Xinje XDPPro project, PLC1: XD5-60T10 (software 3.7.14b 2022-06-24)

PROGRAM 梯形图

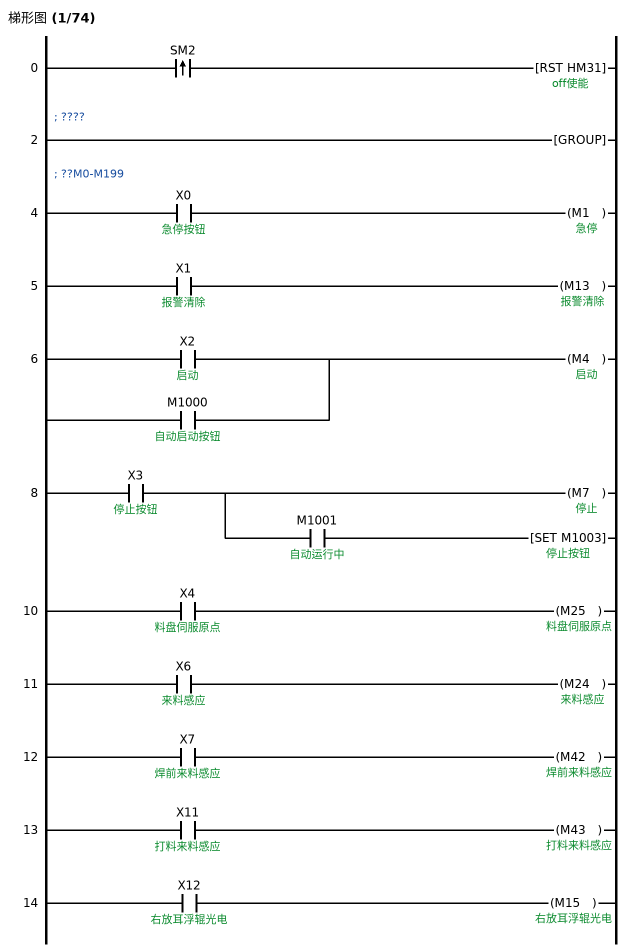
LDP    SM2
RST    HM31	; off使能
; ????
GROUP
; ??M0-M199
LD     X0	; 急停按钮
OUT    M1	; 急停
LD     X1	; 报警清除
OUT    M13	; 报警清除
LD     X2	; 启动
OR     M1000	; 自动启动按钮
OUT    M4	; 启动
LD     X3	; 停止按钮
OUT    M7	; 停止
AND    M1001	; 自动运行中
SET    M1003	; 停止按钮
LD     X4	; 料盘伺服原点
OUT    M25	; 料盘伺服原点
LD     X6	; 来料感应
OUT    M24	; 来料感应
LD     X7	; 焊前来料感应
OUT    M42	; 焊前来料感应
LD     X11	; 打料来料感应
OUT    M43	; 打料来料感应
LD     X12	; 右放耳浮辊光电
OUT    M15	; 右放耳浮辊光电

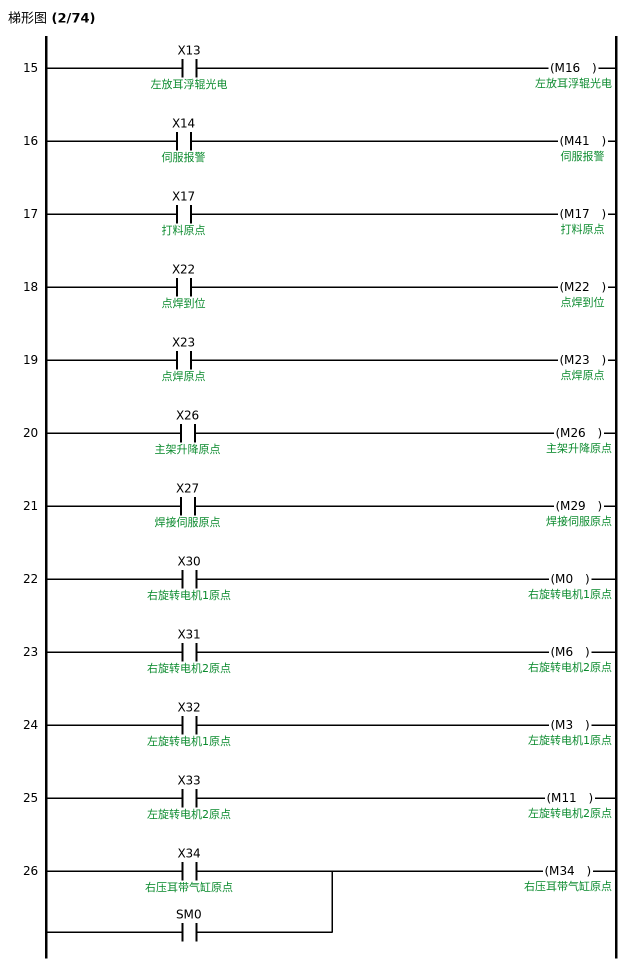
LD     X13	; 左放耳浮辊光电
OUT    M16	; 左放耳浮辊光电
LD     X14	; 伺服报警
OUT    M41	; 伺服报警
LD     X17	; 打料原点
OUT    M17	; 打料原点
LD     X22	; 点焊到位
OUT    M22	; 点焊到位
LD     X23	; 点焊原点
OUT    M23	; 点焊原点
LD     X26	; 主架升降原点
OUT    M26	; 主架升降原点
LD     X27	; 焊接伺服原点
OUT    M29	; 焊接伺服原点
LD     X30	; 右旋转电机1原点
OUT    M0	; 右旋转电机1原点
LD     X31	; 右旋转电机2原点
OUT    M6	; 右旋转电机2原点
LD     X32	; 左旋转电机1原点
OUT    M3	; 左旋转电机1原点
LD     X33	; 左旋转电机2原点
OUT    M11	; 左旋转电机2原点
LD     X34	; 右压耳带气缸原点
OR     SM0
OUT    M34	; 右压耳带气缸原点

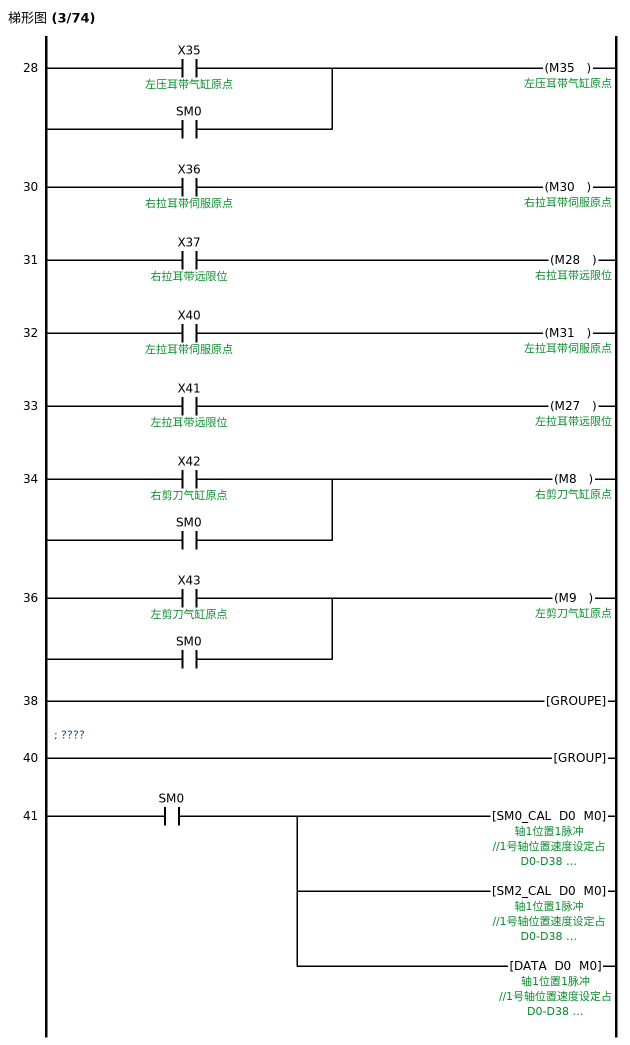
LD     X35	; 左压耳带气缸原点
OR     SM0
OUT    M35	; 左压耳带气缸原点
LD     X36	; 右拉耳带伺服原点
OUT    M30	; 右拉耳带伺服原点
LD     X37	; 右拉耳带远限位
OUT    M28	; 右拉耳带远限位
LD     X40	; 左拉耳带伺服原点
OUT    M31	; 左拉耳带伺服原点
LD     X41	; 左拉耳带远限位
OUT    M27	; 左拉耳带远限位
LD     X42	; 右剪刀气缸原点
OR     SM0
OUT    M8	; 右剪刀气缸原点
LD     X43	; 左剪刀气缸原点
OR     SM0
OUT    M9	; 左剪刀气缸原点
GROUPE
; ????
GROUP
LD     SM0
SM0_CAL D0 M0	; 轴1位置1脉冲   //1号轴位置速度设定占D0-D38 / 右旋转电机1原点
SM2_CAL D0 M0	; 轴1位置1脉冲   //1号轴位置速度设定占D0-D38 / 右旋转电机1原点
DATA   D0 M0	; 轴1位置1脉冲   //1号轴位置速度设定占D0-D38 / 右旋转电机1原点

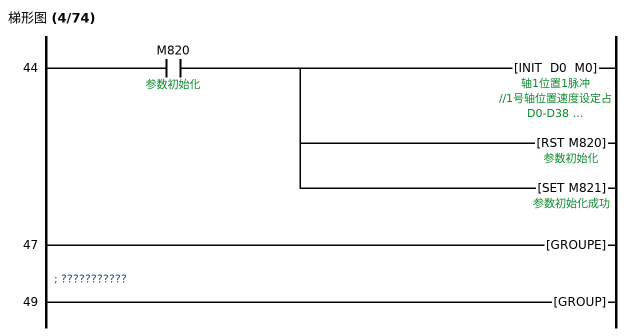
LD     M820	; 参数初始化
INIT   D0 M0	; 轴1位置1脉冲   //1号轴位置速度设定占D0-D38 / 右旋转电机1原点
RST    M820	; 参数初始化
SET    M821	; 参数初始化成功
GROUPE
; ???????????
GROUP

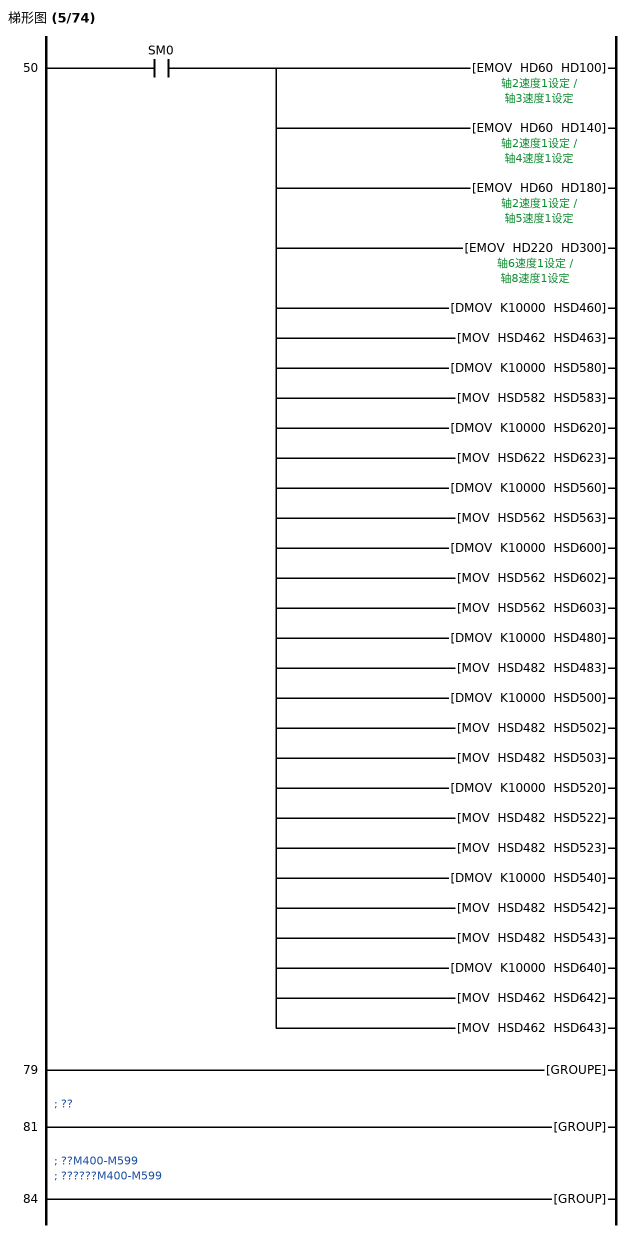
LD     SM0
EMOV   HD60 HD100	; 轴2速度1设定 / 轴3速度1设定
EMOV   HD60 HD140	; 轴2速度1设定 / 轴4速度1设定
EMOV   HD60 HD180	; 轴2速度1设定 / 轴5速度1设定
EMOV   HD220 HD300	; 轴6速度1设定 / 轴8速度1设定
DMOV   K10000 HSD460
MOV    HSD462 HSD463
DMOV   K10000 HSD580
MOV    HSD582 HSD583
DMOV   K10000 HSD620
MOV    HSD622 HSD623
DMOV   K10000 HSD560
MOV    HSD562 HSD563
DMOV   K10000 HSD600
MOV    HSD562 HSD602
MOV    HSD562 HSD603
DMOV   K10000 HSD480
MOV    HSD482 HSD483
DMOV   K10000 HSD500
MOV    HSD482 HSD502
MOV    HSD482 HSD503
DMOV   K10000 HSD520
MOV    HSD482 HSD522
MOV    HSD482 HSD523
DMOV   K10000 HSD540
MOV    HSD482 HSD542
MOV    HSD482 HSD543
DMOV   K10000 HSD640
MOV    HSD462 HSD642
MOV    HSD462 HSD643
GROUPE
; ??
GROUP
; ??M400-M599
; ??????M400-M599
GROUP

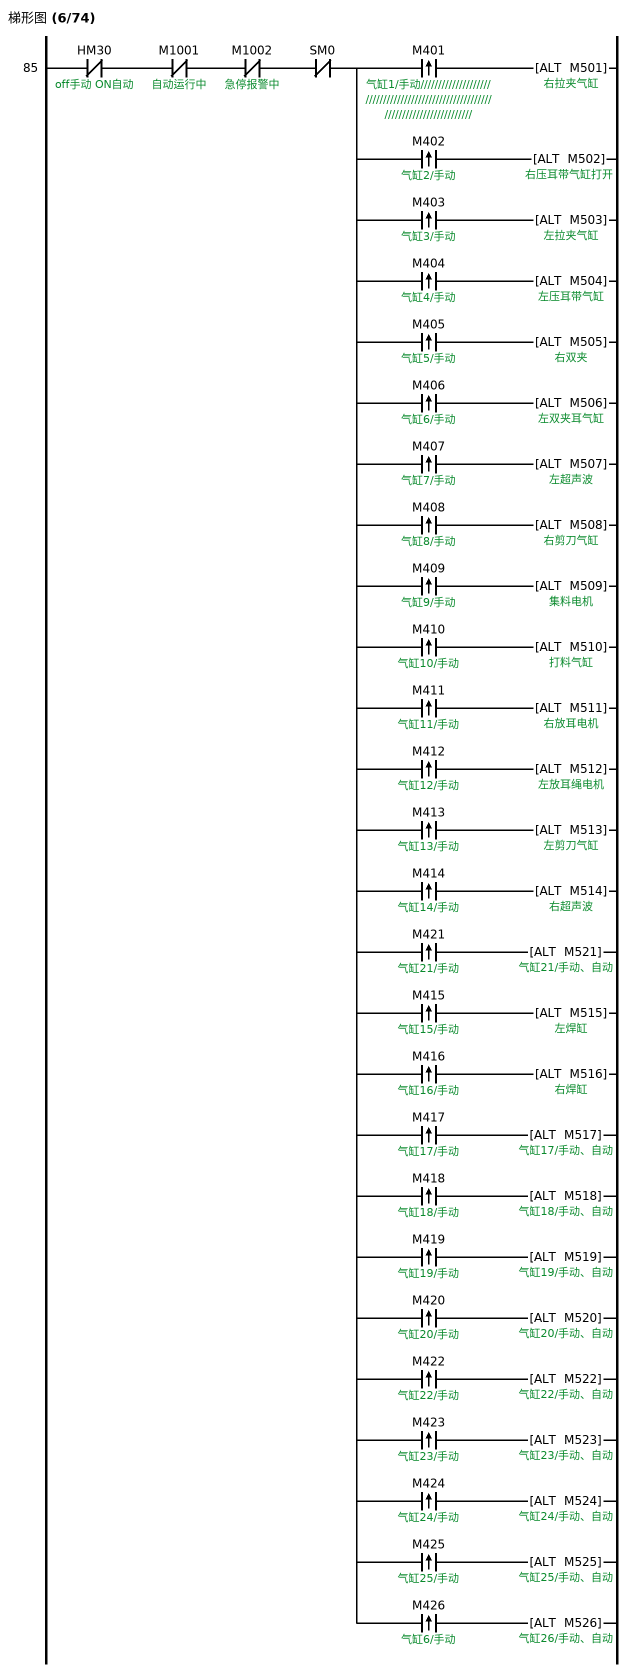
LDI    HM30	; off手动 ON自动
ANI    M1001	; 自动运行中
ANI    M1002	; 急停报警中
ANI    SM0
MPS
ANDP   M401	; 气缸1/手动/////////////////////////////////////////////////////////////////////////////////
ALT    M501	; 右拉夹气缸
MRD
ANDP   M402	; 气缸2/手动
ALT    M502	; 右压耳带气缸打开
MRD
ANDP   M403	; 气缸3/手动
ALT    M503	; 左拉夹气缸
MRD
ANDP   M404	; 气缸4/手动
ALT    M504	; 左压耳带气缸
MRD
ANDP   M405	; 气缸5/手动
ALT    M505	; 右双夹
MRD
ANDP   M406	; 气缸6/手动
ALT    M506	; 左双夹耳气缸
MRD
ANDP   M407	; 气缸7/手动
ALT    M507	; 左超声波
MRD
ANDP   M408	; 气缸8/手动
ALT    M508	; 右剪刀气缸
MRD
ANDP   M409	; 气缸9/手动
ALT    M509	; 集料电机
MRD
ANDP   M410	; 气缸10/手动
ALT    M510	; 打料气缸
MRD
ANDP   M411	; 气缸11/手动
ALT    M511	; 右放耳电机
MRD
ANDP   M412	; 气缸12/手动
ALT    M512	; 左放耳绳电机
MRD
ANDP   M413	; 气缸13/手动
ALT    M513	; 左剪刀气缸
MRD
ANDP   M414	; 气缸14/手动
ALT    M514	; 右超声波
MRD
ANDP   M421	; 气缸21/手动
ALT    M521	; 气缸21/手动、自动
MRD
ANDP   M415	; 气缸15/手动
ALT    M515	; 左焊缸
MRD
ANDP   M416	; 气缸16/手动
ALT    M516	; 右焊缸
MRD
ANDP   M417	; 气缸17/手动
ALT    M517	; 气缸17/手动、自动
MRD
ANDP   M418	; 气缸18/手动
ALT    M518	; 气缸18/手动、自动
MRD
ANDP   M419	; 气缸19/手动
ALT    M519	; 气缸19/手动、自动
MRD
ANDP   M420	; 气缸20/手动
ALT    M520	; 气缸20/手动、自动
MRD
ANDP   M422	; 气缸22/手动
ALT    M522	; 气缸22/手动、自动
MRD
ANDP   M423	; 气缸23/手动
ALT    M523	; 气缸23/手动、自动
MRD
ANDP   M424	; 气缸24/手动
ALT    M524	; 气缸24/手动、自动
MRD
ANDP   M425	; 气缸25/手动
ALT    M525	; 气缸25/手动、自动
MPP
ANDP   M426	; 气缸6/手动
ALT    M526	; 气缸26/手动、自动

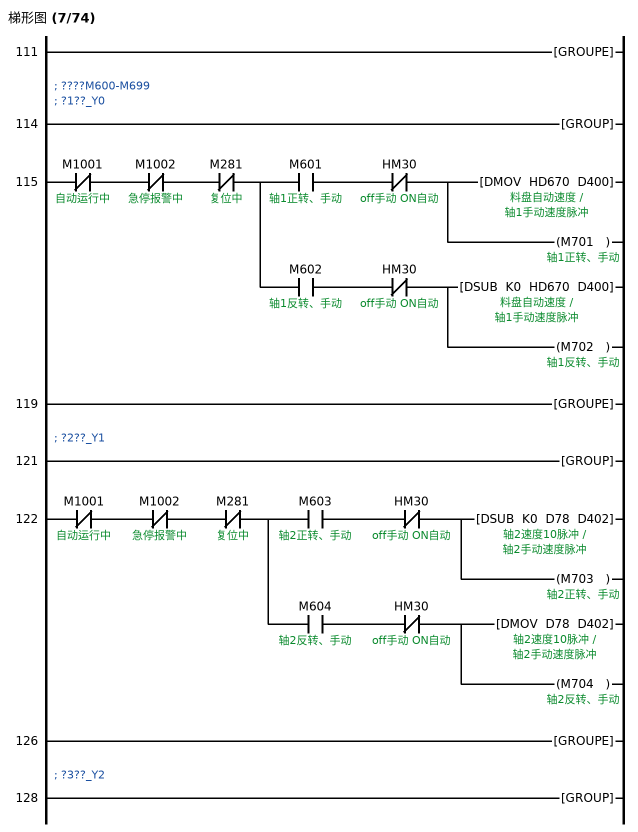
GROUPE
; ????M600-M699
; ?1??_Y0
GROUP
LDI    M1001	; 自动运行中
ANI    M1002	; 急停报警中
ANI    M281	; 复位中
MPS
AND    M601	; 轴1正转、手动
ANI    HM30	; off手动 ON自动
DMOV   HD670 D400	; 料盘自动速度 / 轴1手动速度脉冲
OUT    M701	; 轴1正转、手动
MPP
AND    M602	; 轴1反转、手动
ANI    HM30	; off手动 ON自动
DSUB   K0 HD670 D400	; 料盘自动速度 / 轴1手动速度脉冲
OUT    M702	; 轴1反转、手动
GROUPE
; ?2??_Y1
GROUP
LDI    M1001	; 自动运行中
ANI    M1002	; 急停报警中
ANI    M281	; 复位中
MPS
AND    M603	; 轴2正转、手动
ANI    HM30	; off手动 ON自动
DSUB   K0 D78 D402	; 轴2速度10脉冲 / 轴2手动速度脉冲
OUT    M703	; 轴2正转、手动
MPP
AND    M604	; 轴2反转、手动
ANI    HM30	; off手动 ON自动
DMOV   D78 D402	; 轴2速度10脉冲 / 轴2手动速度脉冲
OUT    M704	; 轴2反转、手动
GROUPE
; ?3??_Y2
GROUP

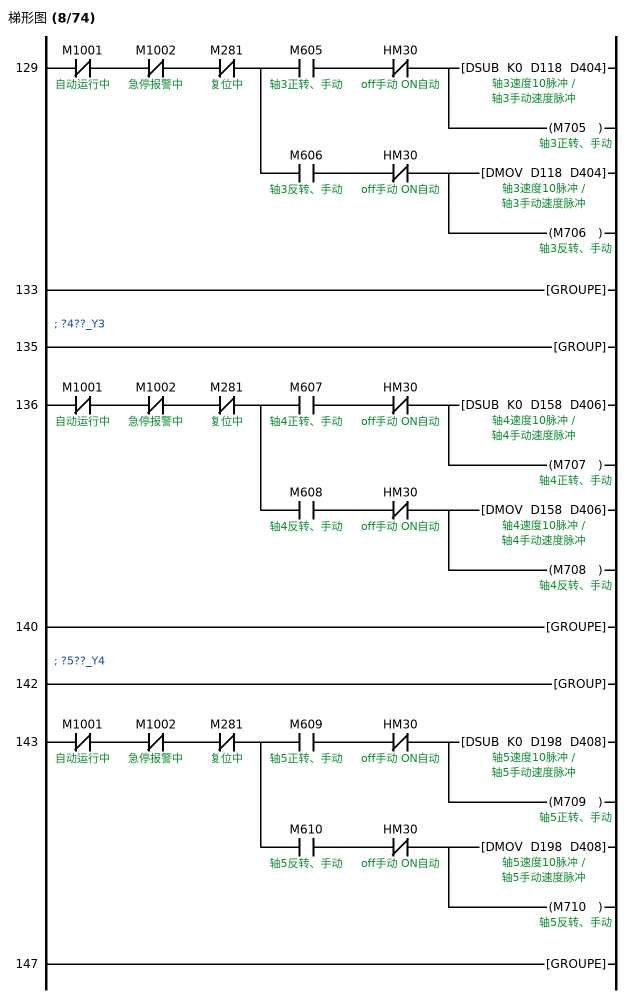
LDI    M1001	; 自动运行中
ANI    M1002	; 急停报警中
ANI    M281	; 复位中
MPS
AND    M605	; 轴3正转、手动
ANI    HM30	; off手动 ON自动
DSUB   K0 D118 D404	; 轴3速度10脉冲 / 轴3手动速度脉冲
OUT    M705	; 轴3正转、手动
MPP
AND    M606	; 轴3反转、手动
ANI    HM30	; off手动 ON自动
DMOV   D118 D404	; 轴3速度10脉冲 / 轴3手动速度脉冲
OUT    M706	; 轴3反转、手动
GROUPE
; ?4??_Y3
GROUP
LDI    M1001	; 自动运行中
ANI    M1002	; 急停报警中
ANI    M281	; 复位中
MPS
AND    M607	; 轴4正转、手动
ANI    HM30	; off手动 ON自动
DSUB   K0 D158 D406	; 轴4速度10脉冲 / 轴4手动速度脉冲
OUT    M707	; 轴4正转、手动
MPP
AND    M608	; 轴4反转、手动
ANI    HM30	; off手动 ON自动
DMOV   D158 D406	; 轴4速度10脉冲 / 轴4手动速度脉冲
OUT    M708	; 轴4反转、手动
GROUPE
; ?5??_Y4
GROUP
LDI    M1001	; 自动运行中
ANI    M1002	; 急停报警中
ANI    M281	; 复位中
MPS
AND    M609	; 轴5正转、手动
ANI    HM30	; off手动 ON自动
DSUB   K0 D198 D408	; 轴5速度10脉冲 / 轴5手动速度脉冲
OUT    M709	; 轴5正转、手动
MPP
AND    M610	; 轴5反转、手动
ANI    HM30	; off手动 ON自动
DMOV   D198 D408	; 轴5速度10脉冲 / 轴5手动速度脉冲
OUT    M710	; 轴5反转、手动
GROUPE

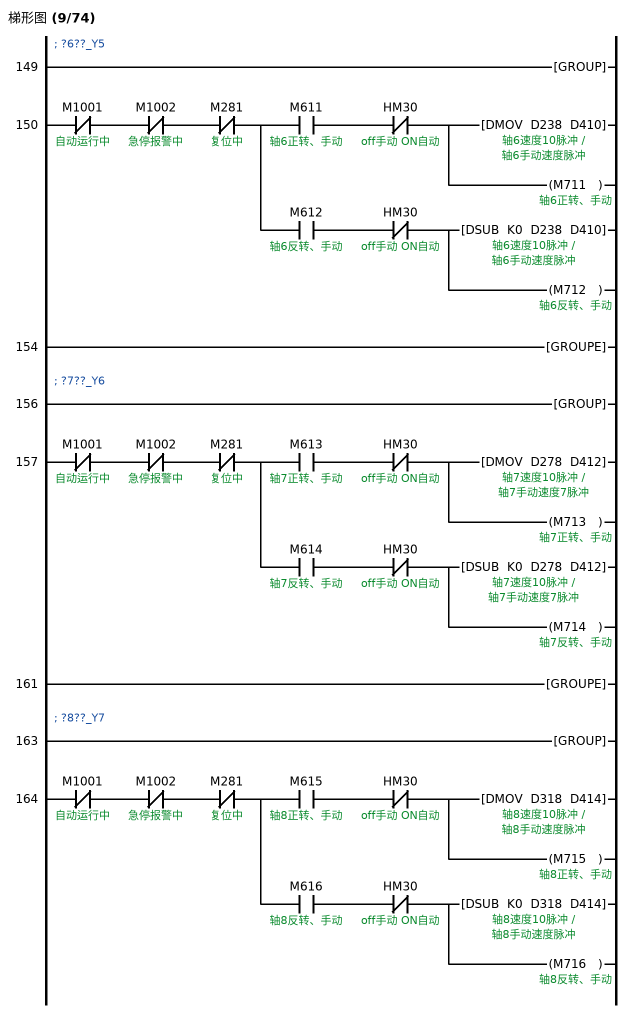
; ?6??_Y5
GROUP
LDI    M1001	; 自动运行中
ANI    M1002	; 急停报警中
ANI    M281	; 复位中
MPS
AND    M611	; 轴6正转、手动
ANI    HM30	; off手动 ON自动
DMOV   D238 D410	; 轴6速度10脉冲 / 轴6手动速度脉冲
OUT    M711	; 轴6正转、手动
MPP
AND    M612	; 轴6反转、手动
ANI    HM30	; off手动 ON自动
DSUB   K0 D238 D410	; 轴6速度10脉冲 / 轴6手动速度脉冲
OUT    M712	; 轴6反转、手动
GROUPE
; ?7??_Y6
GROUP
LDI    M1001	; 自动运行中
ANI    M1002	; 急停报警中
ANI    M281	; 复位中
MPS
AND    M613	; 轴7正转、手动
ANI    HM30	; off手动 ON自动
DMOV   D278 D412	; 轴7速度10脉冲 / 轴7手动速度7脉冲
OUT    M713	; 轴7正转、手动
MPP
AND    M614	; 轴7反转、手动
ANI    HM30	; off手动 ON自动
DSUB   K0 D278 D412	; 轴7速度10脉冲 / 轴7手动速度7脉冲
OUT    M714	; 轴7反转、手动
GROUPE
; ?8??_Y7
GROUP
LDI    M1001	; 自动运行中
ANI    M1002	; 急停报警中
ANI    M281	; 复位中
MPS
AND    M615	; 轴8正转、手动
ANI    HM30	; off手动 ON自动
DMOV   D318 D414	; 轴8速度10脉冲 / 轴8手动速度脉冲
OUT    M715	; 轴8正转、手动
MPP
AND    M616	; 轴8反转、手动
ANI    HM30	; off手动 ON自动
DSUB   K0 D318 D414	; 轴8速度10脉冲 / 轴8手动速度脉冲
OUT    M716	; 轴8反转、手动

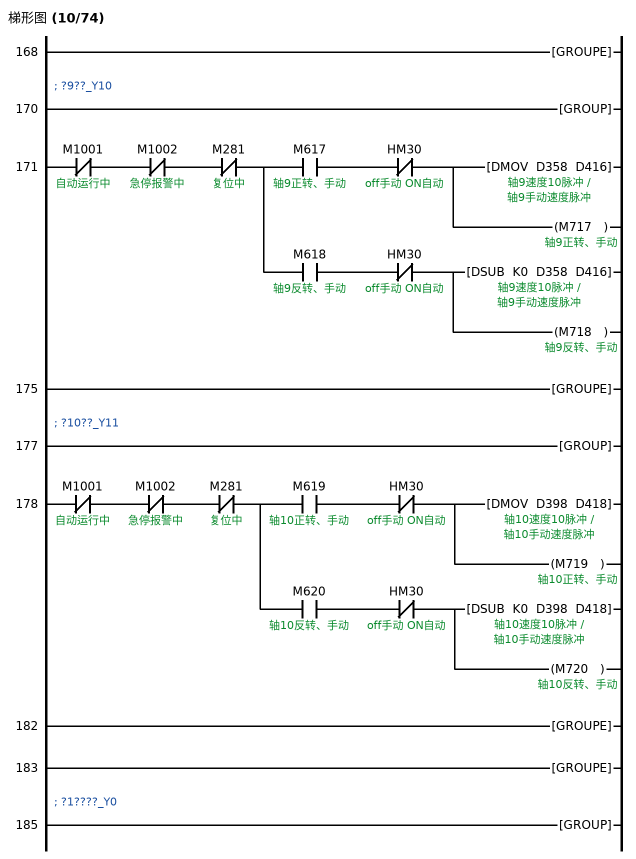
GROUPE
; ?9??_Y10
GROUP
LDI    M1001	; 自动运行中
ANI    M1002	; 急停报警中
ANI    M281	; 复位中
MPS
AND    M617	; 轴9正转、手动
ANI    HM30	; off手动 ON自动
DMOV   D358 D416	; 轴9速度10脉冲 / 轴9手动速度脉冲
OUT    M717	; 轴9正转、手动
MPP
AND    M618	; 轴9反转、手动
ANI    HM30	; off手动 ON自动
DSUB   K0 D358 D416	; 轴9速度10脉冲 / 轴9手动速度脉冲
OUT    M718	; 轴9反转、手动
GROUPE
; ?10??_Y11
GROUP
LDI    M1001	; 自动运行中
ANI    M1002	; 急停报警中
ANI    M281	; 复位中
MPS
AND    M619	; 轴10正转、手动
ANI    HM30	; off手动 ON自动
DMOV   D398 D418	; 轴10速度10脉冲 / 轴10手动速度脉冲
OUT    M719	; 轴10正转、手动
MPP
AND    M620	; 轴10反转、手动
ANI    HM30	; off手动 ON自动
DSUB   K0 D398 D418	; 轴10速度10脉冲 / 轴10手动速度脉冲
OUT    M720	; 轴10反转、手动
GROUPE
GROUPE
; ?1????_Y0
GROUP

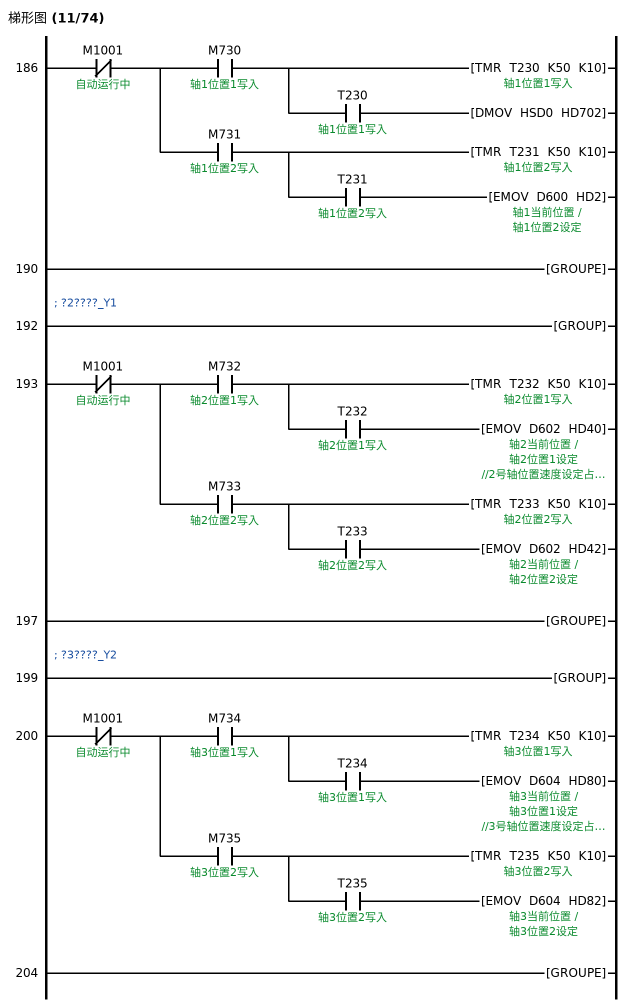
LDI    M1001	; 自动运行中
MPS
AND    M730	; 轴1位置1写入
TMR    T230 K50 K10	; 轴1位置1写入
AND    T230	; 轴1位置1写入
DMOV   HSD0 HD702
MPP
AND    M731	; 轴1位置2写入
TMR    T231 K50 K10	; 轴1位置2写入
AND    T231	; 轴1位置2写入
EMOV   D600 HD2	; 轴1当前位置 / 轴1位置2设定
GROUPE
; ?2????_Y1
GROUP
LDI    M1001	; 自动运行中
MPS
AND    M732	; 轴2位置1写入
TMR    T232 K50 K10	; 轴2位置1写入
AND    T232	; 轴2位置1写入
EMOV   D602 HD40	; 轴2当前位置 / 轴2位置1设定   //2号轴位置速度设定占HD40-HD78
MPP
AND    M733	; 轴2位置2写入
TMR    T233 K50 K10	; 轴2位置2写入
AND    T233	; 轴2位置2写入
EMOV   D602 HD42	; 轴2当前位置 / 轴2位置2设定
GROUPE
; ?3????_Y2
GROUP
LDI    M1001	; 自动运行中
MPS
AND    M734	; 轴3位置1写入
TMR    T234 K50 K10	; 轴3位置1写入
AND    T234	; 轴3位置1写入
EMOV   D604 HD80	; 轴3当前位置 / 轴3位置1设定   //3号轴位置速度设定占HD80-HD118
MPP
AND    M735	; 轴3位置2写入
TMR    T235 K50 K10	; 轴3位置2写入
AND    T235	; 轴3位置2写入
EMOV   D604 HD82	; 轴3当前位置 / 轴3位置2设定
GROUPE

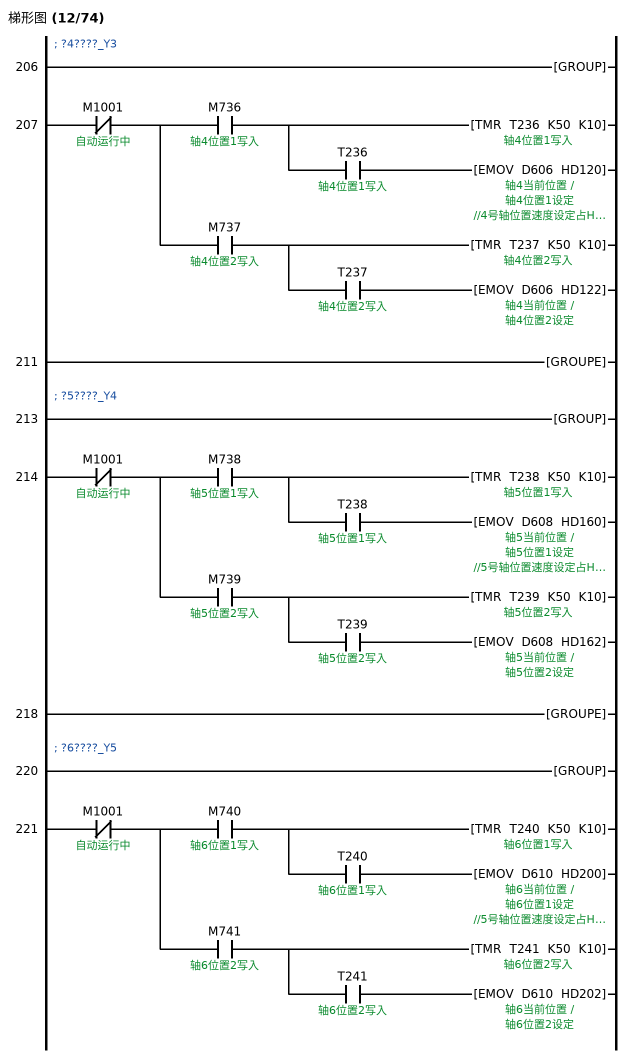
; ?4????_Y3
GROUP
LDI    M1001	; 自动运行中
MPS
AND    M736	; 轴4位置1写入
TMR    T236 K50 K10	; 轴4位置1写入
AND    T236	; 轴4位置1写入
EMOV   D606 HD120	; 轴4当前位置 / 轴4位置1设定   //4号轴位置速度设定占HD120-HD158
MPP
AND    M737	; 轴4位置2写入
TMR    T237 K50 K10	; 轴4位置2写入
AND    T237	; 轴4位置2写入
EMOV   D606 HD122	; 轴4当前位置 / 轴4位置2设定
GROUPE
; ?5????_Y4
GROUP
LDI    M1001	; 自动运行中
MPS
AND    M738	; 轴5位置1写入
TMR    T238 K50 K10	; 轴5位置1写入
AND    T238	; 轴5位置1写入
EMOV   D608 HD160	; 轴5当前位置 / 轴5位置1设定   //5号轴位置速度设定占HD160-HD198
MPP
AND    M739	; 轴5位置2写入
TMR    T239 K50 K10	; 轴5位置2写入
AND    T239	; 轴5位置2写入
EMOV   D608 HD162	; 轴5当前位置 / 轴5位置2设定
GROUPE
; ?6????_Y5
GROUP
LDI    M1001	; 自动运行中
MPS
AND    M740	; 轴6位置1写入
TMR    T240 K50 K10	; 轴6位置1写入
AND    T240	; 轴6位置1写入
EMOV   D610 HD200	; 轴6当前位置 / 轴6位置1设定   //5号轴位置速度设定占HD200-HD238
MPP
AND    M741	; 轴6位置2写入
TMR    T241 K50 K10	; 轴6位置2写入
AND    T241	; 轴6位置2写入
EMOV   D610 HD202	; 轴6当前位置 / 轴6位置2设定

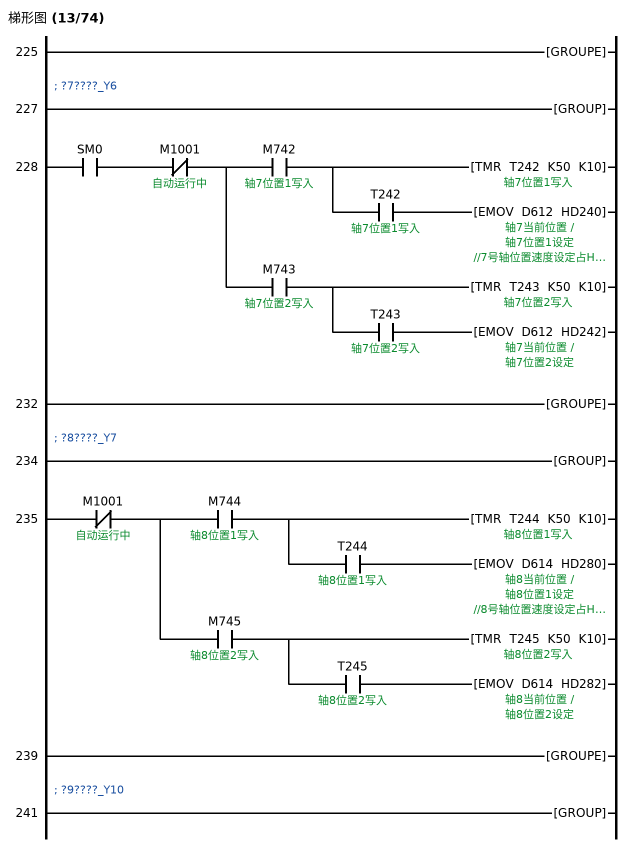
GROUPE
; ?7????_Y6
GROUP
LD     SM0
ANI    M1001	; 自动运行中
MPS
AND    M742	; 轴7位置1写入
TMR    T242 K50 K10	; 轴7位置1写入
AND    T242	; 轴7位置1写入
EMOV   D612 HD240	; 轴7当前位置 / 轴7位置1设定   //7号轴位置速度设定占HD240-HD278
MPP
AND    M743	; 轴7位置2写入
TMR    T243 K50 K10	; 轴7位置2写入
AND    T243	; 轴7位置2写入
EMOV   D612 HD242	; 轴7当前位置 / 轴7位置2设定
GROUPE
; ?8????_Y7
GROUP
LDI    M1001	; 自动运行中
MPS
AND    M744	; 轴8位置1写入
TMR    T244 K50 K10	; 轴8位置1写入
AND    T244	; 轴8位置1写入
EMOV   D614 HD280	; 轴8当前位置 / 轴8位置1设定   //8号轴位置速度设定占HD280-HD318
MPP
AND    M745	; 轴8位置2写入
TMR    T245 K50 K10	; 轴8位置2写入
AND    T245	; 轴8位置2写入
EMOV   D614 HD282	; 轴8当前位置 / 轴8位置2设定
GROUPE
; ?9????_Y10
GROUP

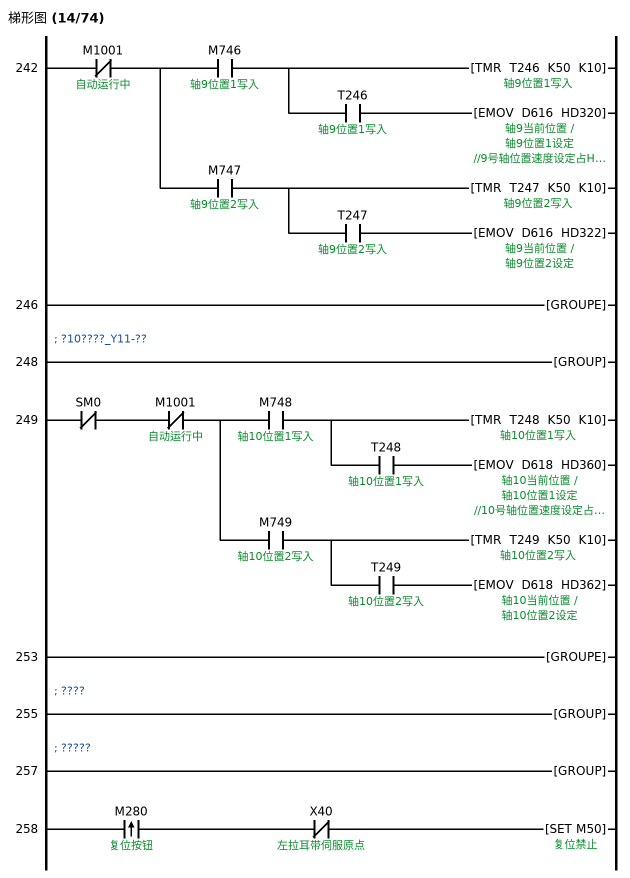
LDI    M1001	; 自动运行中
MPS
AND    M746	; 轴9位置1写入
TMR    T246 K50 K10	; 轴9位置1写入
AND    T246	; 轴9位置1写入
EMOV   D616 HD320	; 轴9当前位置 / 轴9位置1设定   //9号轴位置速度设定占HD320-HD358
MPP
AND    M747	; 轴9位置2写入
TMR    T247 K50 K10	; 轴9位置2写入
AND    T247	; 轴9位置2写入
EMOV   D616 HD322	; 轴9当前位置 / 轴9位置2设定
GROUPE
; ?10????_Y11-??
GROUP
LDI    SM0
ANI    M1001	; 自动运行中
MPS
AND    M748	; 轴10位置1写入
TMR    T248 K50 K10	; 轴10位置1写入
AND    T248	; 轴10位置1写入
EMOV   D618 HD360	; 轴10当前位置 / 轴10位置1设定   //10号轴位置速度设定占HD360-HD398
MPP
AND    M749	; 轴10位置2写入
TMR    T249 K50 K10	; 轴10位置2写入
AND    T249	; 轴10位置2写入
EMOV   D618 HD362	; 轴10当前位置 / 轴10位置2设定
GROUPE
; ????
GROUP
; ?????
GROUP
LDP    M280	; 复位按钮
ANI    X40	; 左拉耳带伺服原点
SET    M50	; 复位禁止

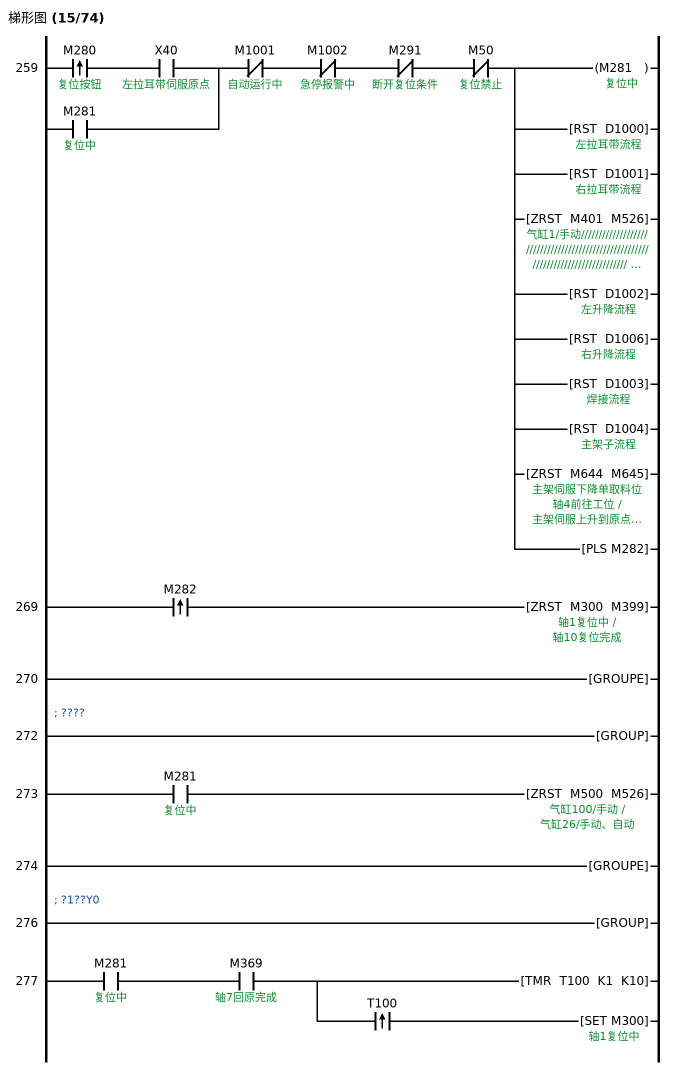
LDP    M280	; 复位按钮
AND    X40	; 左拉耳带伺服原点
OR     M281	; 复位中
ANI    M1001	; 自动运行中
ANI    M1002	; 急停报警中
ANI    M291	; 断开复位条件
ANI    M50	; 复位禁止
OUT    M281	; 复位中
RST    D1000	; 左拉耳带流程
RST    D1001	; 右拉耳带流程
ZRST   M401 M526	; 气缸1/手动///////////////////////////////////////////////////////////////////////////////// / 气缸26/手动、自动
RST    D1002	; 左升降流程
RST    D1006	; 右升降流程
RST    D1003	; 焊接流程
RST    D1004	; 主架子流程
ZRST   M644 M645	; 主架伺服下降单取料位 轴4前往工位 / 主架伺服上升到原点位 轴4前往原点位
PLS    M282
LDP    M282
ZRST   M300 M399	; 轴1复位中 / 轴10复位完成
GROUPE
; ????
GROUP
LD     M281	; 复位中
ZRST   M500 M526	; 气缸100/手动 / 气缸26/手动、自动
GROUPE
; ?1??Y0
GROUP
LD     M281	; 复位中
AND    M369	; 轴7回原完成
TMR    T100 K1 K10
ANDP   T100
SET    M300	; 轴1复位中

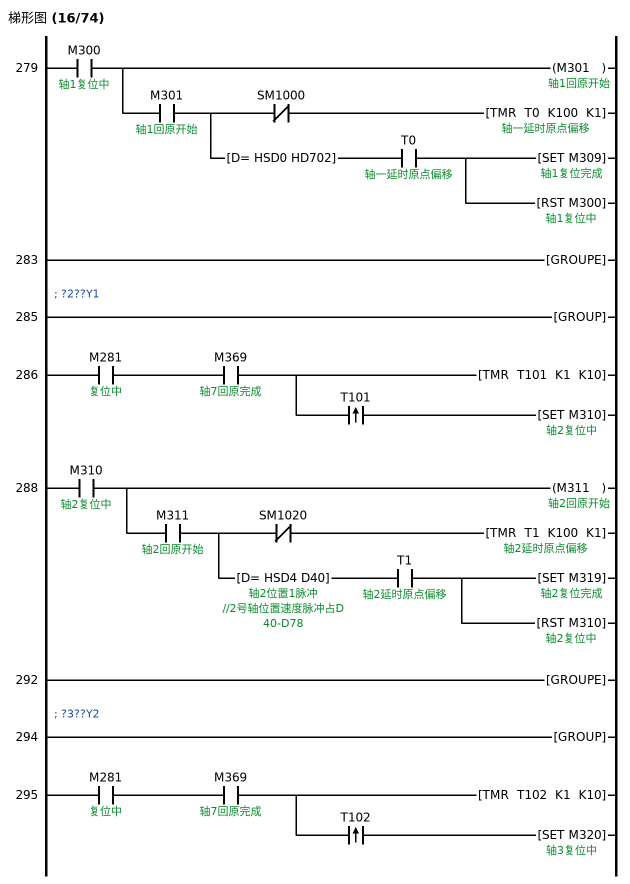
LD     M300	; 轴1复位中
OUT    M301	; 轴1回原开始
AND    M301	; 轴1回原开始
MPS
ANI    SM1000
TMR    T0 K100 K1	; 轴一延时原点偏移
MPP
DAND=  HSD0 HD702
AND    T0	; 轴一延时原点偏移
SET    M309	; 轴1复位完成
RST    M300	; 轴1复位中
GROUPE
; ?2??Y1
GROUP
LD     M281	; 复位中
AND    M369	; 轴7回原完成
TMR    T101 K1 K10
ANDP   T101
SET    M310	; 轴2复位中
LD     M310	; 轴2复位中
OUT    M311	; 轴2回原开始
AND    M311	; 轴2回原开始
MPS
ANI    SM1020
TMR    T1 K100 K1	; 轴2延时原点偏移
MPP
DAND=  HSD4 D40	; 轴2位置1脉冲    //2号轴位置速度脉冲占D40-D78
AND    T1	; 轴2延时原点偏移
SET    M319	; 轴2复位完成
RST    M310	; 轴2复位中
GROUPE
; ?3??Y2
GROUP
LD     M281	; 复位中
AND    M369	; 轴7回原完成
TMR    T102 K1 K10
ANDP   T102
SET    M320	; 轴3复位中

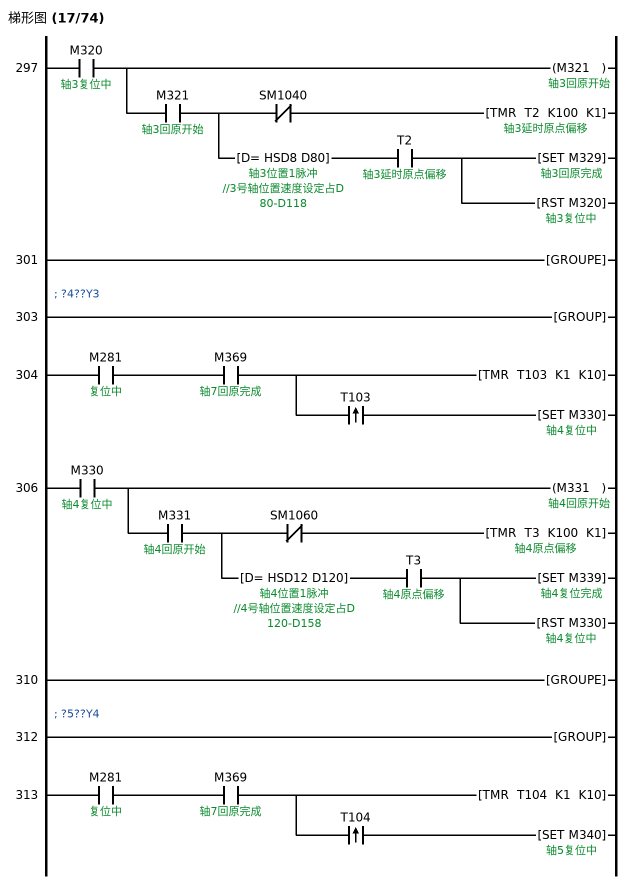
LD     M320	; 轴3复位中
OUT    M321	; 轴3回原开始
AND    M321	; 轴3回原开始
MPS
ANI    SM1040
TMR    T2 K100 K1	; 轴3延时原点偏移
MPP
DAND=  HSD8 D80	; 轴3位置1脉冲   //3号轴位置速度设定占D80-D118
AND    T2	; 轴3延时原点偏移
SET    M329	; 轴3回原完成
RST    M320	; 轴3复位中
GROUPE
; ?4??Y3
GROUP
LD     M281	; 复位中
AND    M369	; 轴7回原完成
TMR    T103 K1 K10
ANDP   T103
SET    M330	; 轴4复位中
LD     M330	; 轴4复位中
OUT    M331	; 轴4回原开始
AND    M331	; 轴4回原开始
MPS
ANI    SM1060
TMR    T3 K100 K1	; 轴4原点偏移
MPP
DAND=  HSD12 D120	; 轴4位置1脉冲   //4号轴位置速度设定占D120-D158
AND    T3	; 轴4原点偏移
SET    M339	; 轴4复位完成
RST    M330	; 轴4复位中
GROUPE
; ?5??Y4
GROUP
LD     M281	; 复位中
AND    M369	; 轴7回原完成
TMR    T104 K1 K10
ANDP   T104
SET    M340	; 轴5复位中

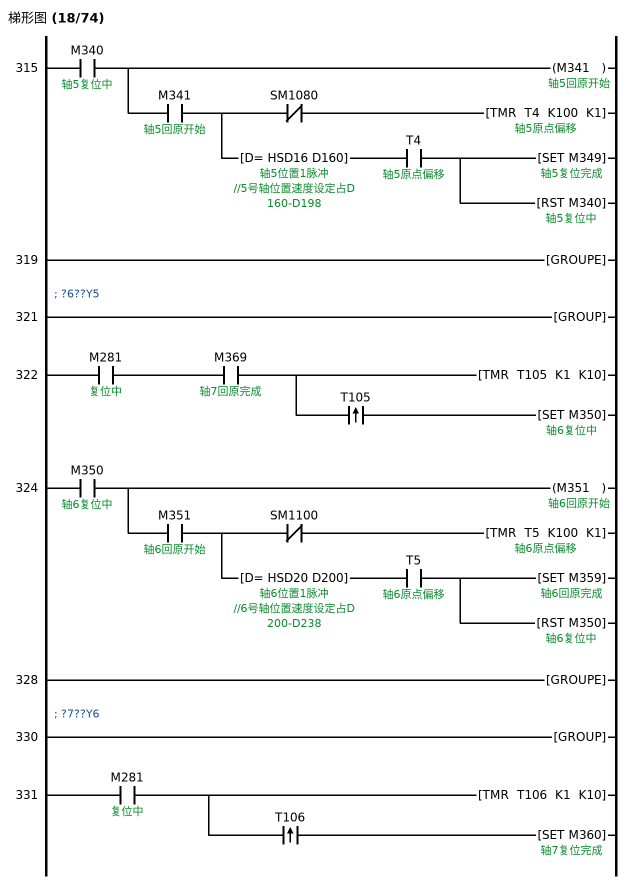
LD     M340	; 轴5复位中
OUT    M341	; 轴5回原开始
AND    M341	; 轴5回原开始
MPS
ANI    SM1080
TMR    T4 K100 K1	; 轴5原点偏移
MPP
DAND=  HSD16 D160	; 轴5位置1脉冲   //5号轴位置速度设定占D160-D198
AND    T4	; 轴5原点偏移
SET    M349	; 轴5复位完成
RST    M340	; 轴5复位中
GROUPE
; ?6??Y5
GROUP
LD     M281	; 复位中
AND    M369	; 轴7回原完成
TMR    T105 K1 K10
ANDP   T105
SET    M350	; 轴6复位中
LD     M350	; 轴6复位中
OUT    M351	; 轴6回原开始
AND    M351	; 轴6回原开始
MPS
ANI    SM1100
TMR    T5 K100 K1	; 轴6原点偏移
MPP
DAND=  HSD20 D200	; 轴6位置1脉冲   //6号轴位置速度设定占D200-D238
AND    T5	; 轴6原点偏移
SET    M359	; 轴6回原完成
RST    M350	; 轴6复位中
GROUPE
; ?7??Y6
GROUP
LD     M281	; 复位中
TMR    T106 K1 K10
ANDP   T106
SET    M360	; 轴7复位完成

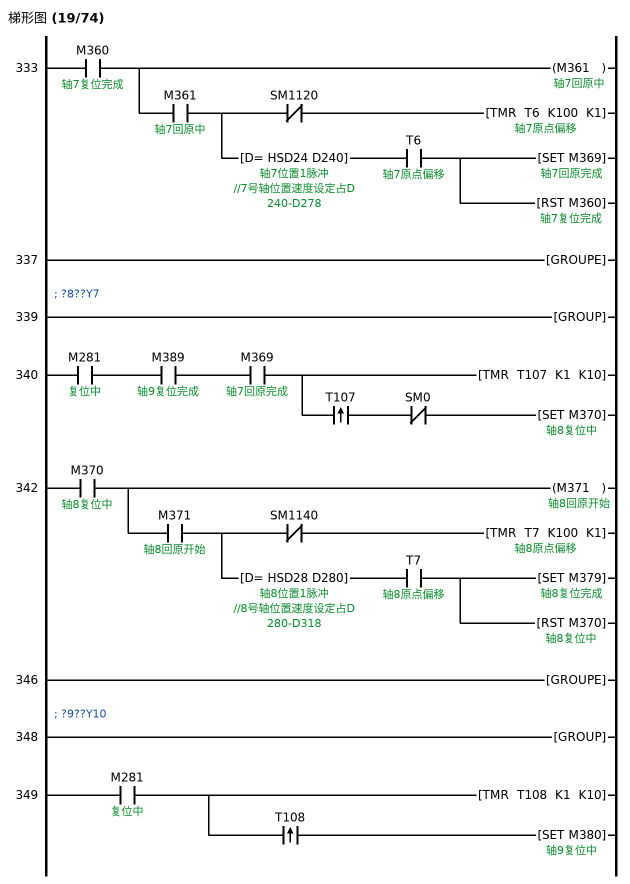
LD     M360	; 轴7复位完成
OUT    M361	; 轴7回原中
AND    M361	; 轴7回原中
MPS
ANI    SM1120
TMR    T6 K100 K1	; 轴7原点偏移
MPP
DAND=  HSD24 D240	; 轴7位置1脉冲   //7号轴位置速度设定占D240-D278
AND    T6	; 轴7原点偏移
SET    M369	; 轴7回原完成
RST    M360	; 轴7复位完成
GROUPE
; ?8??Y7
GROUP
LD     M281	; 复位中
AND    M389	; 轴9复位完成
AND    M369	; 轴7回原完成
TMR    T107 K1 K10
ANDP   T107
ANI    SM0
SET    M370	; 轴8复位中
LD     M370	; 轴8复位中
OUT    M371	; 轴8回原开始
AND    M371	; 轴8回原开始
MPS
ANI    SM1140
TMR    T7 K100 K1	; 轴8原点偏移
MPP
DAND=  HSD28 D280	; 轴8位置1脉冲   //8号轴位置速度设定占D280-D318
AND    T7	; 轴8原点偏移
SET    M379	; 轴8复位完成
RST    M370	; 轴8复位中
GROUPE
; ?9??Y10
GROUP
LD     M281	; 复位中
TMR    T108 K1 K10
ANDP   T108
SET    M380	; 轴9复位中

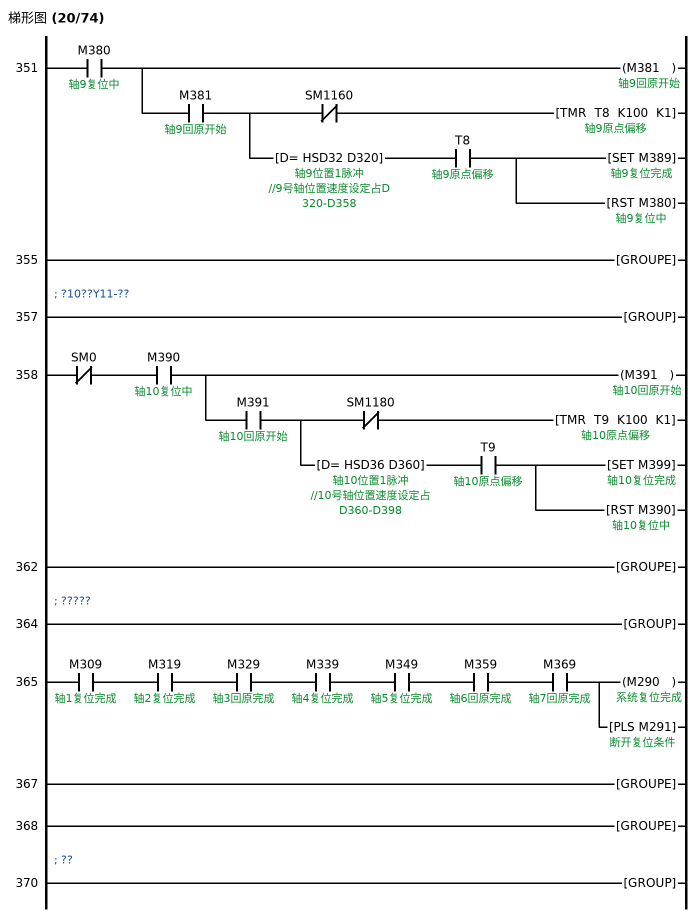
LD     M380	; 轴9复位中
OUT    M381	; 轴9回原开始
AND    M381	; 轴9回原开始
MPS
ANI    SM1160
TMR    T8 K100 K1	; 轴9原点偏移
MPP
DAND=  HSD32 D320	; 轴9位置1脉冲   //9号轴位置速度设定占D320-D358
AND    T8	; 轴9原点偏移
SET    M389	; 轴9复位完成
RST    M380	; 轴9复位中
GROUPE
; ?10??Y11-??
GROUP
LDI    SM0
AND    M390	; 轴10复位中
OUT    M391	; 轴10回原开始
AND    M391	; 轴10回原开始
MPS
ANI    SM1180
TMR    T9 K100 K1	; 轴10原点偏移
MPP
DAND=  HSD36 D360	; 轴10位置1脉冲   //10号轴位置速度设定占D360-D398
AND    T9	; 轴10原点偏移
SET    M399	; 轴10复位完成
RST    M390	; 轴10复位中
GROUPE
; ?????
GROUP
LD     M309	; 轴1复位完成
AND    M319	; 轴2复位完成
AND    M329	; 轴3回原完成
AND    M339	; 轴4复位完成
AND    M349	; 轴5复位完成
AND    M359	; 轴6回原完成
AND    M369	; 轴7回原完成
OUT    M290	; 系统复位完成
PLS    M291	; 断开复位条件
GROUPE
GROUPE
; ??
GROUP

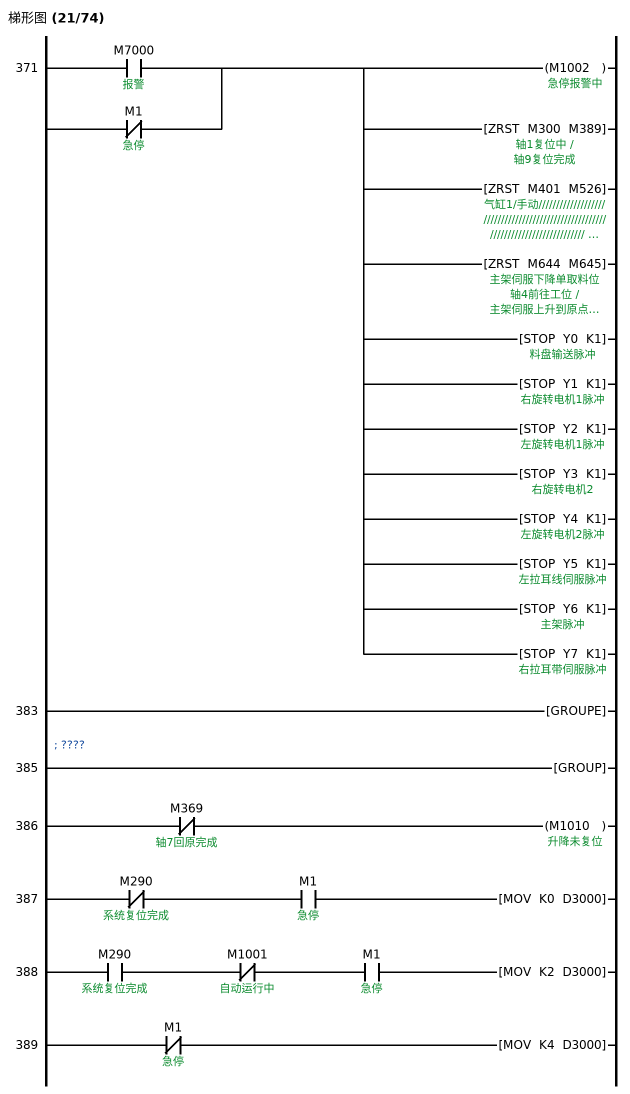
LD     M7000	; 报警
ORI    M1	; 急停
OUT    M1002	; 急停报警中
ZRST   M300 M389	; 轴1复位中 / 轴9复位完成
ZRST   M401 M526	; 气缸1/手动///////////////////////////////////////////////////////////////////////////////// / 气缸26/手动、自动
ZRST   M644 M645	; 主架伺服下降单取料位 轴4前往工位 / 主架伺服上升到原点位 轴4前往原点位
STOP   Y0 K1	; 料盘输送脉冲
STOP   Y1 K1	; 右旋转电机1脉冲
STOP   Y2 K1	; 左旋转电机1脉冲
STOP   Y3 K1	; 右旋转电机2
STOP   Y4 K1	; 左旋转电机2脉冲
STOP   Y5 K1	; 左拉耳线伺服脉冲
STOP   Y6 K1	; 主架脉冲
STOP   Y7 K1	; 右拉耳带伺服脉冲
GROUPE
; ????
GROUP
LDI    M369	; 轴7回原完成
OUT    M1010	; 升降未复位
LDI    M290	; 系统复位完成
AND    M1	; 急停
MOV    K0 D3000
LD     M290	; 系统复位完成
ANI    M1001	; 自动运行中
AND    M1	; 急停
MOV    K2 D3000
LDI    M1	; 急停
MOV    K4 D3000

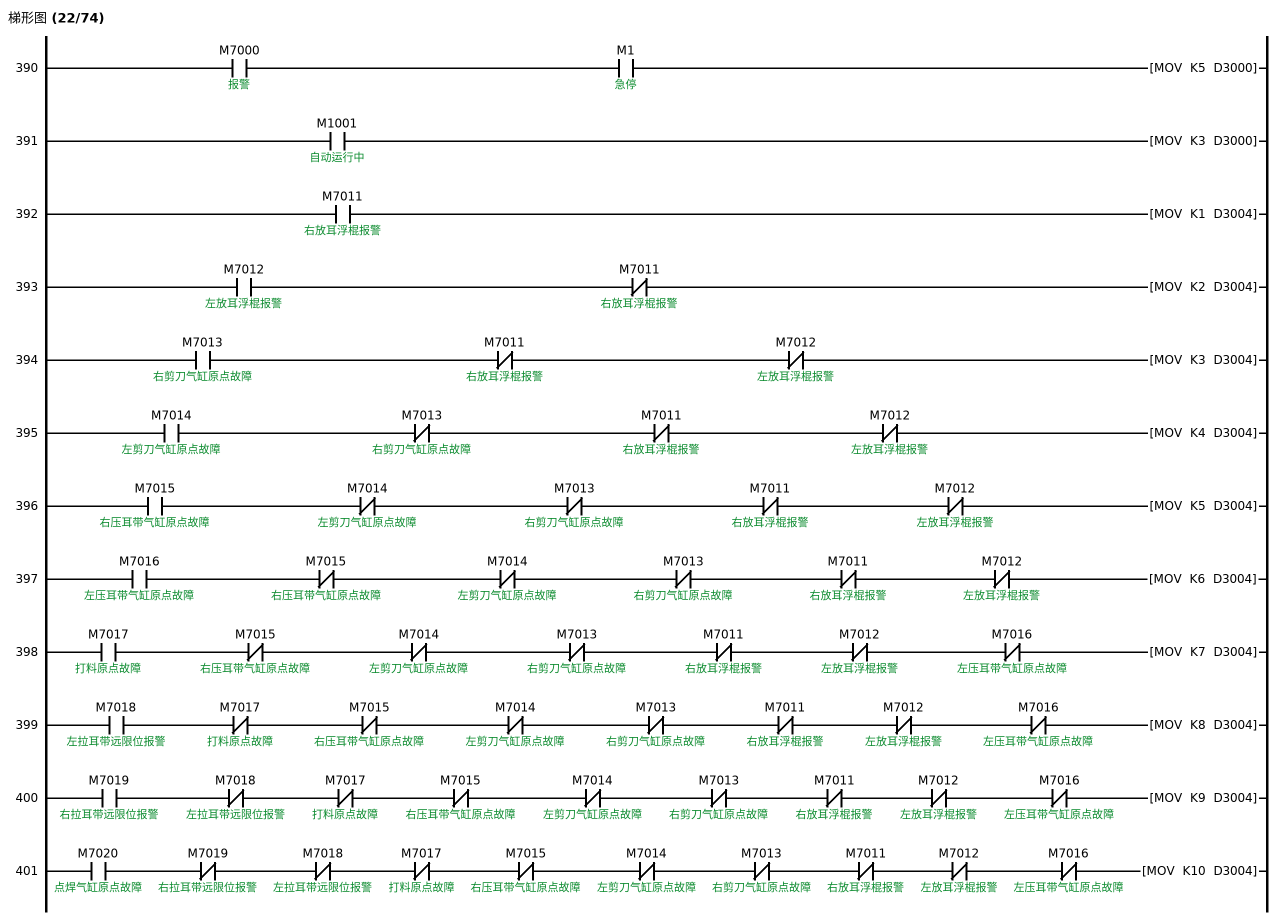
LD     M7000	; 报警
AND    M1	; 急停
MOV    K5 D3000
LD     M1001	; 自动运行中
MOV    K3 D3000
LD     M7011	; 右放耳浮棍报警
MOV    K1 D3004
LD     M7012	; 左放耳浮棍报警
ANI    M7011	; 右放耳浮棍报警
MOV    K2 D3004
LD     M7013	; 右剪刀气缸原点故障
ANI    M7011	; 右放耳浮棍报警
ANI    M7012	; 左放耳浮棍报警
MOV    K3 D3004
LD     M7014	; 左剪刀气缸原点故障
ANI    M7013	; 右剪刀气缸原点故障
ANI    M7011	; 右放耳浮棍报警
ANI    M7012	; 左放耳浮棍报警
MOV    K4 D3004
LD     M7015	; 右压耳带气缸原点故障
ANI    M7014	; 左剪刀气缸原点故障
ANI    M7013	; 右剪刀气缸原点故障
ANI    M7011	; 右放耳浮棍报警
ANI    M7012	; 左放耳浮棍报警
MOV    K5 D3004
LD     M7016	; 左压耳带气缸原点故障
ANI    M7015	; 右压耳带气缸原点故障
ANI    M7014	; 左剪刀气缸原点故障
ANI    M7013	; 右剪刀气缸原点故障
ANI    M7011	; 右放耳浮棍报警
ANI    M7012	; 左放耳浮棍报警
MOV    K6 D3004
LD     M7017	; 打料原点故障
ANI    M7015	; 右压耳带气缸原点故障
ANI    M7014	; 左剪刀气缸原点故障
ANI    M7013	; 右剪刀气缸原点故障
ANI    M7011	; 右放耳浮棍报警
ANI    M7012	; 左放耳浮棍报警
ANI    M7016	; 左压耳带气缸原点故障
MOV    K7 D3004
LD     M7018	; 左拉耳带远限位报警
ANI    M7017	; 打料原点故障
ANI    M7015	; 右压耳带气缸原点故障
ANI    M7014	; 左剪刀气缸原点故障
ANI    M7013	; 右剪刀气缸原点故障
ANI    M7011	; 右放耳浮棍报警
ANI    M7012	; 左放耳浮棍报警
ANI    M7016	; 左压耳带气缸原点故障
MOV    K8 D3004
LD     M7019	; 右拉耳带远限位报警
ANI    M7018	; 左拉耳带远限位报警
ANI    M7017	; 打料原点故障
ANI    M7015	; 右压耳带气缸原点故障
ANI    M7014	; 左剪刀气缸原点故障
ANI    M7013	; 右剪刀气缸原点故障
ANI    M7011	; 右放耳浮棍报警
ANI    M7012	; 左放耳浮棍报警
ANI    M7016	; 左压耳带气缸原点故障
MOV    K9 D3004
LD     M7020	; 点焊气缸原点故障
ANI    M7019	; 右拉耳带远限位报警
ANI    M7018	; 左拉耳带远限位报警
ANI    M7017	; 打料原点故障
ANI    M7015	; 右压耳带气缸原点故障
ANI    M7014	; 左剪刀气缸原点故障
ANI    M7013	; 右剪刀气缸原点故障
ANI    M7011	; 右放耳浮棍报警
ANI    M7012	; 左放耳浮棍报警
ANI    M7016	; 左压耳带气缸原点故障
MOV    K10 D3004

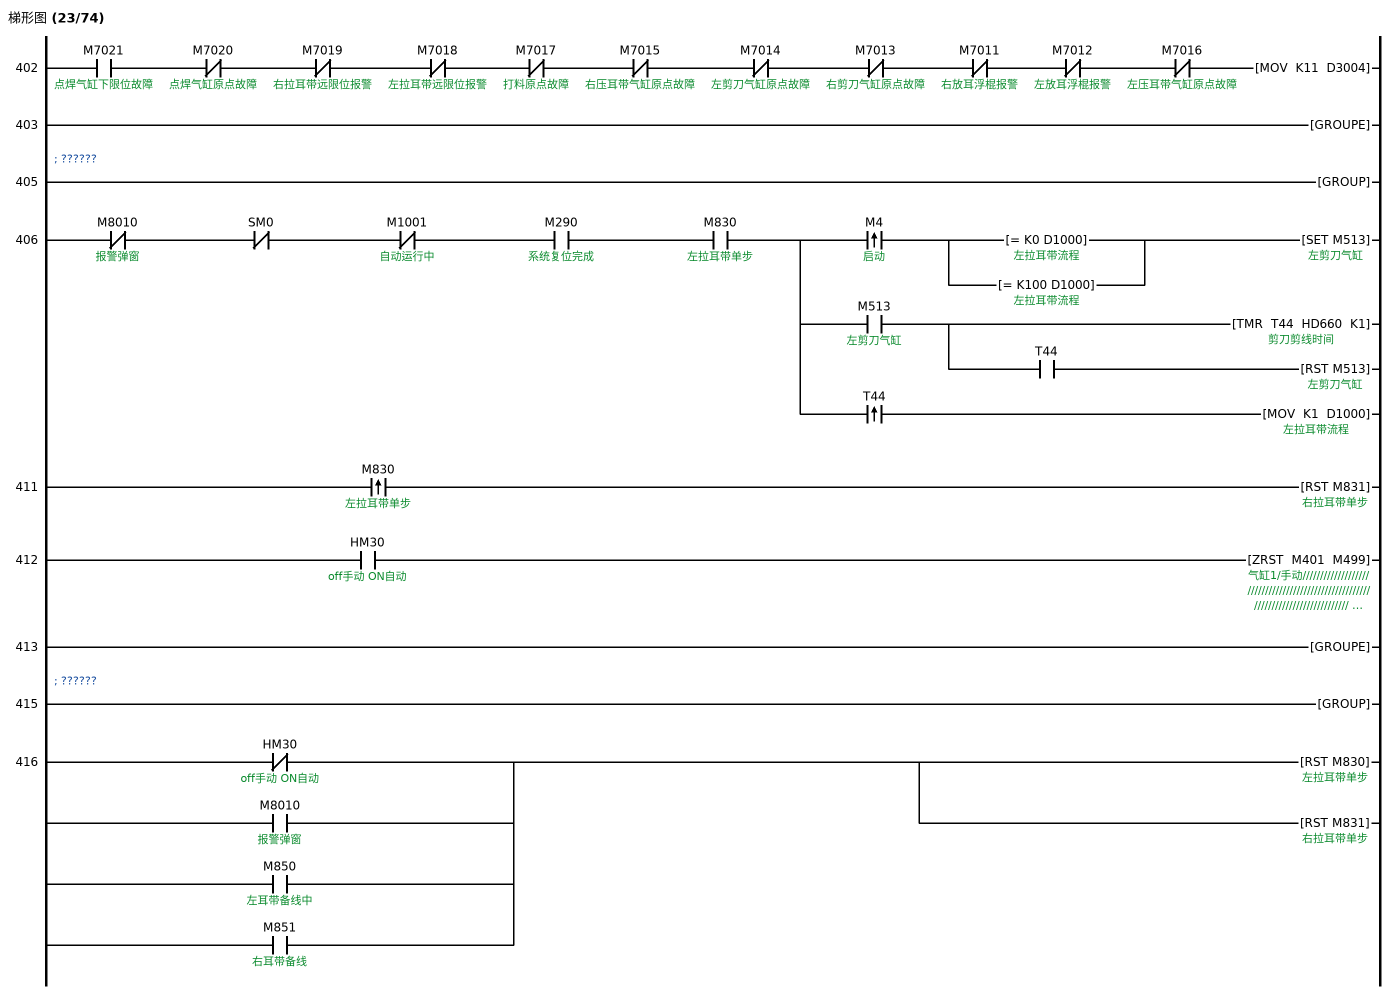
LD     M7021	; 点焊气缸下限位故障
ANI    M7020	; 点焊气缸原点故障
ANI    M7019	; 右拉耳带远限位报警
ANI    M7018	; 左拉耳带远限位报警
ANI    M7017	; 打料原点故障
ANI    M7015	; 右压耳带气缸原点故障
ANI    M7014	; 左剪刀气缸原点故障
ANI    M7013	; 右剪刀气缸原点故障
ANI    M7011	; 右放耳浮棍报警
ANI    M7012	; 左放耳浮棍报警
ANI    M7016	; 左压耳带气缸原点故障
MOV    K11 D3004
GROUPE
; ??????
GROUP
LDI    M8010	; 报警弹窗
ANI    SM0
ANI    M1001	; 自动运行中
AND    M290	; 系统复位完成
AND    M830	; 左拉耳带单步
MPS
ANDP   M4	; 启动
LD=    K0 D1000	; 左拉耳带流程
OR=    K100 D1000	; 左拉耳带流程
ANB
SET    M513	; 左剪刀气缸
MRD
AND    M513	; 左剪刀气缸
TMR    T44 HD660 K1	; 剪刀剪线时间
AND    T44
RST    M513	; 左剪刀气缸
MPP
ANDP   T44
MOV    K1 D1000	; 左拉耳带流程
LDP    M830	; 左拉耳带单步
RST    M831	; 右拉耳带单步
LD     HM30	; off手动 ON自动
ZRST   M401 M499	; 气缸1/手动///////////////////////////////////////////////////////////////////////////////// / 气缸99/手动
GROUPE
; ??????
GROUP
LDI    HM30	; off手动 ON自动
OR     M8010	; 报警弹窗
OR     M850	; 左耳带备线中
OR     M851	; 右耳带备线
RST    M830	; 左拉耳带单步
RST    M831	; 右拉耳带单步

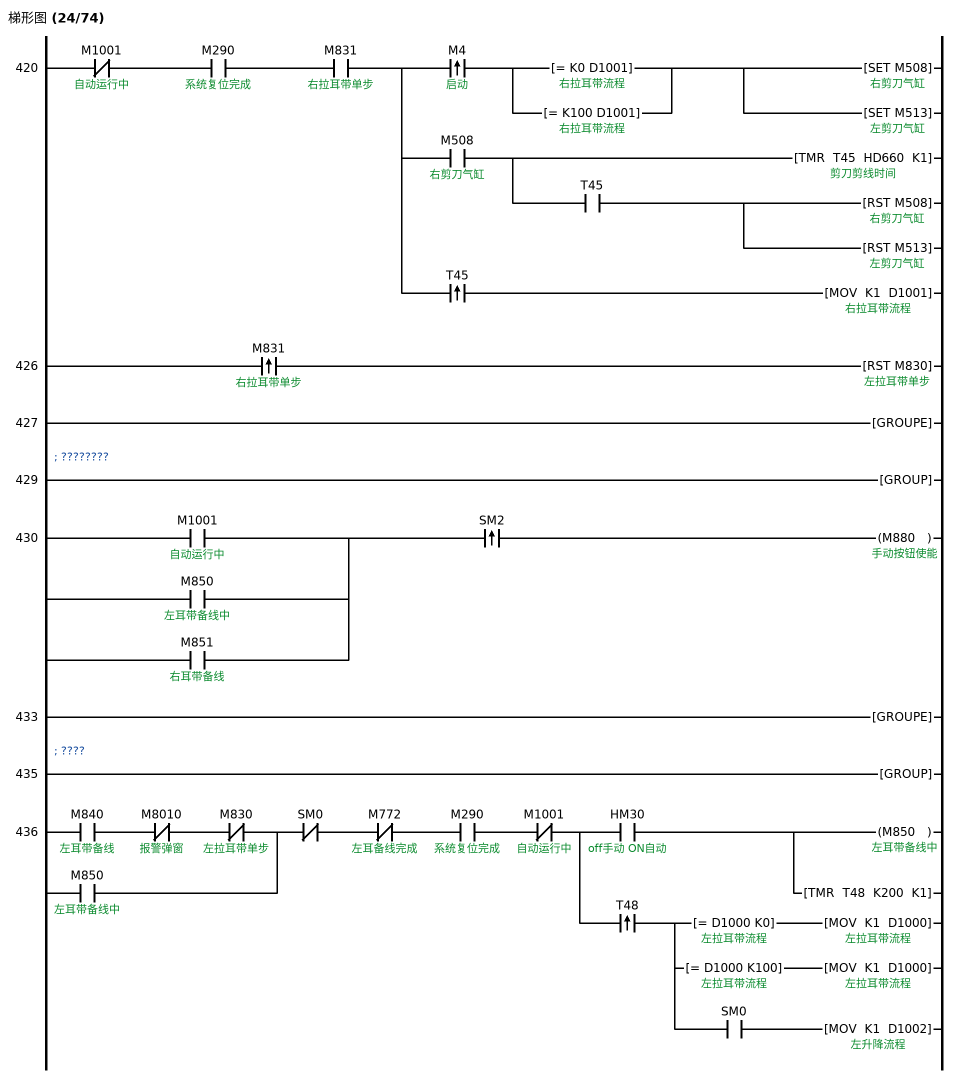
LDI    M1001	; 自动运行中
AND    M290	; 系统复位完成
AND    M831	; 右拉耳带单步
MPS
ANDP   M4	; 启动
LD=    K0 D1001	; 右拉耳带流程
OR=    K100 D1001	; 右拉耳带流程
ANB
SET    M508	; 右剪刀气缸
SET    M513	; 左剪刀气缸
MRD
AND    M508	; 右剪刀气缸
TMR    T45 HD660 K1	; 剪刀剪线时间
AND    T45
RST    M508	; 右剪刀气缸
RST    M513	; 左剪刀气缸
MPP
ANDP   T45
MOV    K1 D1001	; 右拉耳带流程
LDP    M831	; 右拉耳带单步
RST    M830	; 左拉耳带单步
GROUPE
; ????????
GROUP
LD     M1001	; 自动运行中
OR     M850	; 左耳带备线中
OR     M851	; 右耳带备线
ANDP   SM2
OUT    M880	; 手动按钮使能
GROUPE
; ????
GROUP
LD     M840	; 左耳带备线
ANI    M8010	; 报警弹窗
ANI    M830	; 左拉耳带单步
OR     M850	; 左耳带备线中
ANI    SM0
ANI    M772	; 左耳备线完成
AND    M290	; 系统复位完成
ANI    M1001	; 自动运行中
MPS
AND    HM30	; off手动 ON自动
OUT    M850	; 左耳带备线中
TMR    T48 K200 K1
MPP
ANDP   T48
MPS
AND=   D1000 K0	; 左拉耳带流程
MOV    K1 D1000	; 左拉耳带流程
MRD
AND=   D1000 K100	; 左拉耳带流程
MOV    K1 D1000	; 左拉耳带流程
MPP
AND    SM0
MOV    K1 D1002	; 左升降流程

